TYPE ST_HS_Zustand :
STRUCT
	Betrieb					: BOOL;
	Betrieb_Anford_KW		: BOOL;
	Betrieb_Anford_WW		: BOOL;

	Kommunikation			: BOOL;

	Stoerung				: BOOL;
	Stoerung_Code			: WORD;

	Warnung					: BOOL;
	Warnung_Code			: WORD;

	Status					: SINT;
END_STRUCT
END_TYPE

(* stored: Version 1.1.0.1, ProductVersion 3.1.4024.9
   DUT ST_HS_Zustand: Id {271eb4ce-347a-4eb4-8487-5c2a1779080a} *)
